# EPICS autosave request: FOFBApp/Db/FOFBAcq_settings.req
$(P)$(R)$(ACQ_NAME)SamplesPre-SP
$(P)$(R)$(ACQ_NAME)SamplesPost-SP
$(P)$(R)$(ACQ_NAME)Shots-SP
$(P)$(R)$(ACQ_NAME)Channel-Sel
$(P)$(R)$(ACQ_NAME)UpdateTime-SP
$(P)$(R)$(ACQ_NAME)Trigger-Sel
$(P)$(R)$(ACQ_NAME)TriggerRep-Sel
$(P)$(R)$(ACQ_NAME)TriggerDataThres-SP
$(P)$(R)$(ACQ_NAME)TriggerDataPol-Sel
$(P)$(R)$(ACQ_NAME)TriggerDataSel-SP
$(P)$(R)$(ACQ_NAME)TriggerDataHyst-SP
$(P)$(R)$(ACQ_NAME)TriggerHwDly-SP
$(P)$(R)$(ACQ_NAME)TriggerRep-Sel
$(P)$(R)$(ACQ)$(ARRAY_NAME)ArrayDataWvf
$(P)$(R)$(ACQ)$(ARRAY_NAME)ArrayData
$(P)$(R)$(ACQ)$(ARRAY_NAME)ArrayDataSeq
